TYPE ParCode : 
STRUCT
    sRemoteHost                :T_IPv4Addr;  //扫描枪IP地址
    sRemotePot                  :UINT;  //端口号
    TimeOut:		               INT:=5;	//扫码超时时间


END_STRUCT
END_TYPE

(* stored: Version 1.1.0.1, ProductVersion 3.1.4024.9
   DUT ParCode: Id {dbc21ca4-b23e-4e47-9bf9-e62924b08720} *)
